{attribute 'linkalways'} 
{attribute 'no_explicit_call' := 'This FB is a CLASS and must be accessed using methods or properties'}
{attribute 'enable_dynamic_creation'}
FUNCTION_BLOCK FINAL XOR_LINT EXTENDS Node
VAR
	in1 : _LINT(0);
	in2 : _LINT(0);
	out : _LINT(0);
END_VAR

METHOD PUBLIC Clone : I_Node
VAR
	pNode : POINTER TO XOR_LINT;
END_VAR
pNode := __NEW(XOR_LINT);
Clone := pNode^;
END_METHOD

METHOD FB_init : BOOL
VAR_INPUT
	bInitRetains : BOOL; // if TRUE, the retain variables are initialized (warm start / cold start)
	bInCopyCode : BOOL;  // if TRUE, the instance afterwards gets moved into the copy code (online change)
END_VAR
AddInput('in1',THIS^.in1);
AddInput('in2',THIS^.in2);
AddOutput('out', THIS^.out);
END_METHOD

METHOD PROTECTED OnExecute
VAR
END_VAR
out.Value := in1.Value XOR in2.Value;
END_METHOD

END_FUNCTION_BLOCK

(* stored: Version 1.1.0.1, ProductVersion 3.1.4024.15
   POU XOR_LINT: Id {158d4ec9-6907-4b47-af29-963b313fa969}, SpecialFunc None
   Folder Constructor: Id {94dd713a-cbf6-4edc-a60a-323335067ac6}
   Method Clone: Id {b4772e8f-8d0f-4828-9c6f-a9acd5493a03}
   Method FB_init: Id {ff8112ff-5c8f-4836-9692-fec000c38d86}
   Method OnExecute: Id {bda217a2-2909-4e33-8998-d321d86a339d} *)
